// TIA Portal V16 export
// export: Created 2022-09-01T13:58:51.2485369Z, ExportSetting WithDefaults, DisplayName Totally Integrated Automation Portal, DisplayVersion V16, DisplayName TIA Portal Version Control Interface, DisplayVersion V16, DisplayName TIA Portal Openness, DisplayVersion V16, DisplayName STEP 7 Professional, DisplayVersion V16, DisplayName STEP 7 Safety, DisplayVersion V16, DisplayName WinCC Advanced, DisplayVersion V16
FUNCTION "Proc_Analog_Press_Filt2" : Void   // FC19, LAD
{ S7_Optimized_Access := 'TRUE' }
VERSION : 0.1
// stored: AutoNumber true, IsIECCheckEnabled false, SetENOAutomatically false, UDAEnableTagReadback false
   VAR_OUTPUT
      Pressão_em_Bar : Real;
   END_VAR
   VAR_TEMP
      "Pressão_em_%" : Real;
   END_VAR
BEGIN

REGION Network 1
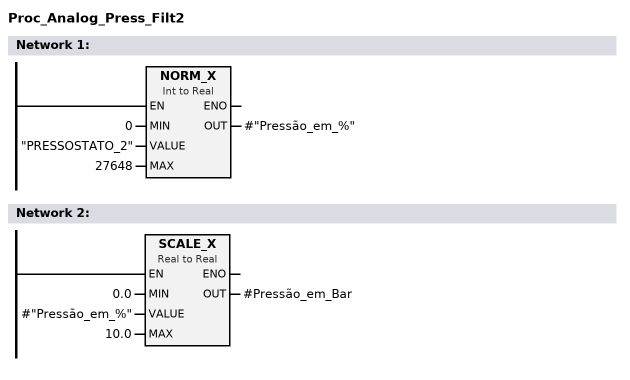
   RUNG wire#powerrail
      { S7_Templates := "[SrcType := Int, DestType := Real]"; S7_GenerateENO := "TRUE" } Normalize(min := 0, value := "PRESSOSTATO_2", max := 27648, out => #"Pressão_em_%")
   END_RUNG
   // the same network as SCL:
   #"Pressão_em_%" := NORM_X(MIN := 0, VALUE := "PRESSOSTATO_2", MAX := 27648);
END_REGION

REGION Network 2
   RUNG wire#powerrail
      { S7_Templates := "[SrcType := Real, DestType := Real]"; S7_GenerateENO := "TRUE" } Scale(min := 0.0, value := #"Pressão_em_%", max := 10.0, out => #Pressão_em_Bar)
   END_RUNG
   // the same network as SCL:
   #Pressão_em_Bar := SCALE_X(MIN := 0.0, VALUE := #"Pressão_em_%", MAX := 10.0);
END_REGION
END_FUNCTION
